FUNCTION_BLOCK FB_GantryXYZ EXTENDS FB_PackML_BaseModule 
VAR
    // Sub module definitions here

    // List of sub modules
    ipSubModules_Init : ARRAY[1..Parameters_PackML_Base.MAX_NO_OF_SUBMODULES] OF I_PackML_BaseModule := [];

    // Component definitions here
    AxisX       		: FB_Component_BasicAxis 		:= (Name := 'AxisX');
    AxisY    			: FB_Component_BasicAxis 		:= (Name := 'AxisY');
	AxisZ				: FB_Component_BasicAxis		:= (Name := 'AxisZ');
    GantryCylinder		: FB_GantryXYCylinder			:= (Name := 'Cylinder');
    //Alarms for this module
    GantryAlarms : ARRAY[1..GANTRY_ALARM_COUNT] OF FB_TcAlarm;

	//IO
	LimitSwitchX :BOOL;
	LimitSwitchY :BOOL;
	LimitSwitchZ :BOOL;

	HomeComplete :BOOL;
	
	//resets


END_VAR

VAR CONSTANT
    GANTRY_ALARM_COUNT : INT := 5;
END_VAR


METHOD PROTECTED Aborting
VAR
	i				: UDINT;
	SubModulesReady : BOOL := TRUE;
END_VAR
CASE SequenceState OF
    0:
        NoStateTasksToComplete := FALSE;
        SequenceState          := SequenceState + 10;
    10:
		AxisX.Disable();
		SequenceState := SequenceState + 10;
	20:

		StateTasksComplete := TRUE;
END_CASE

SUPER^.Aborting();
END_METHOD

METHOD PROTECTED Clearing
VAR
	i				: UDINT;
	SubModulesReady : BOOL := TRUE;
END_VAR

VAR_INST
	SoEResetAxis1 : FB_SoEReset;
	ResetAxis1 :	MC_Reset;
END_VAR
CASE SequenceState OF
    0:
        NoStateTasksToComplete := FALSE;
        SequenceState          := SequenceState + 10;
    10:
		//Reset any alarms that get latched
//		GantryAlarms[E_Gantry.AlarmMessage].Clear(0,0);		
//		GantryAlarms[E_Gantry.InfoMessage].Clear(0,0);
//		GantryAlarms[E_Gantry.InitReferenceEvent].Clear(0,0);
//		GantryAlarms[E_Gantry.StartTimeout].Clear(0,0);
//		GantryAlarms[E_Gantry.WarnMessage].Clear(0,0);
//		AxisX.Reset();
//		AxisY.Reset();
//		AxisZ.Reset();



//		AxisX.Reset();

		SoEResetAxis1(Axis := AxisX.Axis);
		SoEResetAxis1.Execute := TRUE;	
		
		ResetAxis1(Axis:=AxisX.Axis);
		ResetAxis1.Execute := TRUE;
		
		
		SequenceState := SequenceState + 10;
	20:
	
		SequenceState := SequenceState + 10;
30: 

		IF NOT ResetSafety() THEN
			ResetSafety();
		ELSE
			SequenceState := SequenceState + 10;	
		END_IF	
    40:

        // Enable here
		// AxisX.Enable();
		// AxisY.Enable();
		// AxisZ.Enable();

        // Check enabled here
		// IF AxisX.Enabled AND AxisY.Enabled AND AxisZ.Enabled THEN
			// SequenceState := SequenceState + 10;
		// END_IF
		
		SequenceState := SequenceState + 10;
		
    50:
        StateTasksComplete := TRUE;
		
END_CASE

SUPER^.Clearing();
END_METHOD

METHOD PROTECTED CreateEvents
VAR_INPUT
END_VAR
// Add your event creation here
F_CreateAllEventsInClass(Alarms     := GantryAlarms,
                         ClassSize  := SIZEOF(TC_EVENTS.Gantry),
                         pInitEvent := ADR(TC_EVENTS.Gantry.InitReferenceEvent),
                         Prefix     := _Name);

// Super call to base
SUPER^.CreateEvents();
END_METHOD

METHOD CuttingBoxFiveSides : BOOL

VAR_INST
	Step : INT ;	
END_VAR



(*
	F			H
	|			|
D---+-----------+---C
	|			|
	|			| 
B---+-----------+---A
	|			|
	E			G
*)
	CASE Step OF
		
		0:  

//Print Info
			
			Trace('Start Cutting Box Five Sides');


			AxisX.MoveVelocity(1,0);
			
			
			Step := Step + 10;	

		10:	//Set Speed

//			AxisX.Velocity := 10; 
//			AxisY.Velocity := 10;
//			AxisZ.Velocity := 5;
			
			Step := Step + 160;

//		20:	//Positioning Motion to A
   			
//			AxisX.MoveAbsolute(0,0);
//			AxisY.MoveAbsolute(250,0);		
			
//			Step := Step + 10; 
		
//		30: //Set Cutting Height
			
//			AxisZ.MoveAbsolute(-30,0);
			
//			Step := Step + 10;

//		40: //Cutting Motion from A to B
			
//			AxisX.MoveAbsolute(500,0);		
			
//			Step := Step + 10;
		
//		50: //Return from Cutting Height 
			
//			AxisZ.MoveAbsolute(50,0);

//			Step := Step + 10;
		
//		60: //Positioning Motion from B to C
			
//			AxisX.MoveAbsolute(0,0);
//			AxisY.MoveAbsolute(50,0);
	
//			Step := Step + 10;

//		70: //Set Cutting Height
		
//			AxisZ.MoveAbsolute(0,0);

//			Step := Step + 10;

//		80: //Cutting Motion from C to D
			
//			AxisX.MoveAbsolute(500,0);
//			AxisY.MoveAbsolute(50,0);

//			Step := Step + 10;

//		90: //Return from Cutting Height 
			
//			AxisZ.MoveAbsolute(50,0);
			
//			Step := Step + 10;

//		100: //Positioning Motion from D to E
			
//			AxisX.MoveAbsolute(450,0);
//			AxisY.MoveAbsolute(300,0);

//			Step := Step + 10;
		
//		110: //Set Cutting Height 	
			
//			AxisZ.MoveAbsolute(0,0);
	
//			Step := Step + 10;

//		120: //Cutting Motion from E to F

//			AxisX.MoveAbsolute(450,0);
//			AxisY.MoveAbsolute(0,0);
			
//			Step := Step + 10;

//		130: //Return from Cutting Height 

//			AxisZ.MoveAbsolute(50,0);
			
//			Step := Step + 10;

//		140: //Positioning Motion from F to G

//			AxisX.MoveAbsolute(50,0);
//			AxisY.MoveAbsolute(300,0);

//			Step := Step + 10;

//		150: //Cutting Motion from G to H
  
//			AxisX.MoveAbsolute(50,0);
//			AxisY.MoveAbsolute(0,0);

//			Step := Step + 10;

//		160: //Return from Cutting Height 
	
//			AxisZ.MoveAbsolute(50,0);

//			Step := Step + 10;

		170: 

//Return to ZERO
////			AxisX.MoveAbsolute(0,0);
//			AxisY.MoveAbsolute(0,0);
			CuttingBoxFiveSides := TRUE;
			Step := 0;
			Trace('Box Five Sides is Cut');
		
			

		

			
	END_CASE
END_METHOD

METHOD CyclicLogic
VAR_INPUT
END_VAR
IF NOT _InitComplete THEN
    _InitComplete := Initialize();
    RETURN;
END_IF

SUPER^.CyclicLogic();

//Set the current alarm severity for this module
_CurrentAlarmSeverity := F_GetMaxSeverityRaised(Alarms := GantryAlarms, CurrentSeverity := _CurrentAlarmSeverity);

//Simulate Alarm Messaging
END_METHOD

METHOD PROTECTED Execute
CASE _CurrentMode OF

	//=================================PRODUCTION MODE==================================
	E_PMLUnitMode.ePMLUnitMode_Production:
		CASE SequenceState OF
			0:
				NoStateTasksToComplete := FALSE;
				
				IF NOT CuttingBoxFiveSides() THEN
					CuttingBoxFiveSides();	
				ELSE
					SequenceState := SequenceState + 10;
				END_IF		
				
			10:		
				StateTasksComplete := TRUE;
				StateComplete();
			END_CASE

	//=================================MAINTENANCE & MANUAL MODE==================================
	E_PMLUnitMode.ePMLUnitMode_Maintenance, E_PMLUnitMode.ePMLUnitMode_Manual:
		;
END_CASE
END_METHOD

METHOD PROTECTED HMIPermissions
//General Mode Based Monitoring and handling of HMI control
CASE _CurrentMode OF
   
 E_PMLUnitMode.ePMLUnitMode_Production:
        CASE _CurrentState OF
            E_PMLState.ePMLState_Stopped:
				AllowHMIControl(ThisModuleOnly := FALSE);
            E_PMLState.ePMLState_Idle:
				AllowHMIControl(ThisModuleOnly := FALSE);
            E_PMLState.ePMLState_Suspended:
         		AllowHMIControl(ThisModuleOnly := FALSE);
            E_PMLState.ePMLState_Execute:
            	AllowHMIControl(ThisModuleOnly := FALSE); 
            E_PMLState.ePMLState_Aborted:
                AllowHMIControl(ThisModuleOnly := FALSE); 
            E_PMLState.ePMLState_Held:
                AllowHMIControl(ThisModuleOnly := FALSE); 
            E_PMLState.ePMLState_Complete:
          		AllowHMIControl(ThisModuleOnly := FALSE); 
        END_CASE
		
    E_PMLUnitMode.ePMLUnitMode_Manual:
        AllowHMIControl(ThisModuleOnly := FALSE); 
	E_PMLUnitMode.ePMLUnitMode_Maintenance:
        AllowHMIControl(ThisModuleOnly := FALSE); 
END_CASE
END_METHOD

METHOD Homing : BOOL

VAR_INST
	Step : INT ;	
END_VAR
CASE Step OF
		
		0: 
			Trace('Enable');
			AxisX.Enable();
		   //AxisX.MoveVelocity(5,0);
			Step := Step + 10; 
		10:
//			Trace('Move Relative');
//			IF IO.DI4 = FALSE THEN
//				AxisX.Home();
//				Step := Step + 10;
//			END_IF
			
//			IF AxisX.Busy = FALSE THEN
//				Step := Step + 10;
//			END_IF
			
			Step := Step + 10;

	
		20:	
			

			Homing := TRUE;
			Step := 0;	

	END_CASE
END_METHOD

//! @summary Basic module initialization logic
METHOD PROTECTED Initialize : BOOL;
VAR
    i                        : UDINT;
    varInfo                  : __SYSTEM.VAR_INFO;
    AllSubUnitsInitialized   : BOOL := TRUE;
    AllComponentsInitialized : BOOL := TRUE;
END_VAR

//! @description This method is called by <c>CyclicLogic()</c> as required
Initialize := FALSE;
CASE DescendantSequenceState OF
    0:
		RegisterComponent(AxisX);
		RegisterComponent(AxisY);	
		RegisterComponent(AxisZ);	
		RegisterComponent(GantryCylinder);
		
        _LogModeChanges         := FALSE;
        _LogStateChanges        := FALSE;
        DescendantSequenceState := DescendantSequenceState + 10;
    10:
        DescendantSequenceState := DescendantSequenceState + 10;
    20:
        //Copy Mode names
        FOR i := 1 TO 3 DO
            ModeNames[i] := F_UnitModeToString(UDINT_TO_DINT(i));
        END_FOR

        DescendantSequenceState := DescendantSequenceState + 10;
    30:
        //Call the Super
        IF SUPER^.Initialize() THEN
            DescendantSequenceState := DescendantSequenceState + 10;
        END_IF
    40:
        Initialize := TRUE;
END_CASE
END_METHOD

METHOD ResetSafety : BOOL
VAR_INST
	Step : INT ;	
	SafetyTimer :TON;
	SafetyTimerTrigger :R_TRIG;
END_VAR
SafetyTimer(IN:= Step > 0 AND NOT SafetyTimer.Q, PT:= T#500MS);

CASE Step OF
		
		0:  // Reset group or waits
			Trace('Timer Initialize');
			Step := Step + 10;
			
		10: //If necessary reset group
		
			GVL_Safety.ErrorAck := (GVL_Safety.ComError OR GVL_Safety.FBError OR GVL_Safety.SafeError); 
		
			IF GVL_Safety.ErrorAck OR SafetyTimer.Q THEN 
				Step := Step + 10;
			END_IF

		20: //Wait for the signal propagation
			IF SafetyTimer.Q THEN
				GVL_Safety.ErrorAck := FALSE;
				Step := Step + 10;
			END_IF
		
		30: //Check FB errors
			IF GVL_Safety.FBError OR (NOT GVL_Safety.SAFETY_Permission) THEN
				GVL_Safety.RestartFBs_TSG := TRUE;
			END_IF
			
			Step := Step + 10;
			
		40: //Wait for the signal propagation
		
			IF SafetyTimer.Q THEN
				GVL_Safety.RestartFBs_TSG := FALSE;
				Step := Step + 10;
			END_IF	
			
		50: //If necessary reset the AX5805
			;
			
		60: //Wait for the signal propagation

			IF SafetyTimer.Q THEN
				
			
			
				IF GVL_Safety.SAFETY_Permission AND 
					NOT (GVL_Safety.ComError OR GVL_Safety.FBError OR GVL_Safety.SafeError) 
				
					THEN
						Step := 0;
						ResetSafety := TRUE;
					ELSE
						Step := 0;
						ResetSafety := FALSE;
				END_IF
			
			END_IF
		
		ELSE
		
		Step := 0;	

END_CASE
END_METHOD

METHOD PROTECTED Resetting
VAR
	i				: UDINT;
	SubModulesReady : BOOL := TRUE;
END_VAR
CASE _CurrentMode OF

	//=================================PRODUCTION MODE==================================
	E_PMLUnitMode.ePMLUnitMode_Production:
		CASE SequenceState OF
			0:
				NoStateTasksToComplete := TRUE;
				
				IF NOT Homing() THEN
					Homing();
				ELSE
					SequenceState := SequenceState + 10;	
				END_IF		
				
			10:		
				StateTasksComplete := TRUE;
				SUPER^.Resetting();
		END_CASE

	//=================================MAINTENANCE & MANUAL MODE==================================
	E_PMLUnitMode.ePMLUnitMode_Maintenance, E_PMLUnitMode.ePMLUnitMode_Manual:
		;
END_CASE
END_METHOD

END_FUNCTION_BLOCK

(* stored: Version 1.1.0.1, ProductVersion 3.1.4024.15
   POU FB_GantryXYZ: Id {474e1990-f731-0ed9-052c-42626742a38f}, SpecialFunc None
   Folder MyMethods: Id {d166ca9d-f57a-4d88-ac90-142e5eb5d488}
   Folder States: Id {8df42c9b-c051-49f1-9767-900503632339}
   Method Aborting: Id {5476dfef-6652-4e6b-8928-3724a50553de}
   Method Clearing: Id {9be5800b-bdc3-471f-9b7d-42ef121d5c77}
   Method CreateEvents: Id {40e5a283-7f33-033f-0879-cc11ecabc43d}
   Method CuttingBoxFiveSides: Id {391386b3-3ac4-4fc7-a2a1-1d79f5676796}
   Method CyclicLogic: Id {0cfbfa67-40d6-05d6-0515-ef1c50353a78}
   Method Execute: Id {895d1ef9-5e85-47dd-a8bf-b32885837641}
   Method HMIPermissions: Id {a7a517c4-9176-4ef6-9045-d889c05c8a21}
   Method Homing: Id {7cf726af-0fa2-4719-9f55-f55ebcdc06af}
   Method Initialize: Id {ba85f303-ffbe-03ad-229b-3741bd93e6e2}
   Method ResetSafety: Id {6bac4035-16f4-4bf2-95a7-9f0b204a82b7}
   Method Resetting: Id {e7a01217-de28-430f-aeef-f83d9f1b6f0d} *)
